FUNCTION_BLOCK FB_RealControlBox IMPLEMENTS I_ControlBox
VAR_INPUT
END_VAR
VAR_OUTPUT
END_VAR
VAR
END_VAR

METHOD Joystick
VAR_INPUT
	eMode 	: E_Mode;
	eStatus : E_Status;
END_VAR
VAR_OUTPUT
	fJoystickY : LREAL;
END_VAR
END_METHOD

METHOD Lamps 
VAR_INPUT
	eMode 	: E_Mode;
	eStatus : E_Status;
END_VAR
// To Do LAB #12
END_METHOD

METHOD ModeSelector 
VAR_INPUT
END_VAR
VAR_OUTPUT
	eMode : E_Mode;
END_VAR
// To Do LAB #12
END_METHOD

METHOD PushButtons
VAR_INPUT
	eMode 	: E_Mode;
	eStatus : E_Status;
END_VAR
VAR_OUTPUT
	bStart : BOOL;
	bStop : BOOL;
END_VAR
END_METHOD

END_FUNCTION_BLOCK

(* stored: Version 1.1.0.1, ProductVersion 3.1.4024.10
   POU FB_RealControlBox: Id {37de488e-61db-47f0-ae9a-a602c45471dd}, SpecialFunc None
   Method Joystick: Id {969d1bf9-8f4a-4ed0-b706-e8d8185bf738}
   Method Lamps: Id {4fdeda89-2fc2-4bda-9219-00e0aed099ce}
   Method ModeSelector: Id {c1118847-ecf0-4ef4-a589-62e6a17557ee}
   Method PushButtons: Id {d7dda8b1-708c-4ae4-b6f1-5856535cda99} *)
